// TwinCAT 3 PLC project CapSorter
// ProgramVersion: 3.1.4026.19
// libraries:
//   Tc2_Standard, * (Beckhoff Automation GmbH)
//   Tc2_System, * (Beckhoff Automation GmbH)
//   TcEventLogger, * (Beckhoff Automation Poland)
// project tree:
//   GVLs/ GVL.TcGVL, GVL_Checks.TcGVL, GVL_Communication.TcGVL, GVL_ErrorHandling.TcGVL, GVL_IO.TcGVL, GVL_Recipe.TcGVL, GVL_StandAloneUnit.TcGVL, GVL_VIS.TcGVL
//   / PlcTask.TcTTO
//   POUs/ FB_DigitalInput.TcPOU, FB_DigitalOutput.TcPOU, MAIN.TcPOU
// (motion and I/O tree: see PLC project programplc)
// real-time tasks:
//   TASK MainTask: cycle T#3ms, priority 20, ADS port 350
//   TASK SafetyTask: cycle T#10ms, priority 22, ADS port 351
//   TASK WeightTask: cycle T#2ms, priority 19, ADS port 354
//   TASK PlcTask: cycle T#10ms, priority 21, ADS port 355
//   TASK TaskToRefreshEAP: cycle T#1ms, priority 12, ADS port 301
// variable links:

CONFIGURATION CapSorter
    RESOURCE PLC ON TwinCAT3
        TASK PlcTask(INTERVAL := T#10ms, PRIORITY := 21);
        PROGRAM MAIN WITH PlcTask : MAIN;
    END_RESOURCE
END_CONFIGURATION

// ---- GVLs/GVL.TcGVL
{attribute 'qualified_only'}
VAR_GLOBAL
	iRunningMode								: INT	:= 1;					// Pozniej zastanowic sie gdzie to zostawic
END_VAR

// ---- GVLs/GVL_Checks.TcGVL
{attribute 'qualified_only'}
VAR_GLOBAL PERSISTENT
	dCheckBounds					: DINT;			// Licznik przekroczen zakresu indexow, np. tablic
	dCheckDivDInt					: DINT;			// Licznik prob dzielenia Dint przez 0
	dCheckDivLInt					: DINT; 		// Licznik prob dzielenia LInt przez 0
	dCheckDivLReal					: DINT; 		// Licznik prob dzielenia LREAL przez 0
	dCheckDivReal					: DINT; 		// Licznik prob dzielenia REAL przez 0
	dCheckRangeSigned				: DINT;			// Licznik przekroczen liczby znakowej
	dCheckRangeUnsigned				: DINT; 		// Licznik przekroczen liczby bezznakowej
END_VAR

// ---- GVLs/GVL_Communication.TcGVL
VAR_GLOBAL
//	stWrite				AT%MB0		: ST_Communication;			//Wysyłane zmienne do BottleUnboxer
//	stRead				AT%I*		: ST_Communication;			//Odczytane zmienne z BottleUnboxer

	// Sygnały pomocnicze
	bEnable									: BOOL;
	bCycleStart								: BOOL;
	bCycleStop								: BOOL;
	bCycleReset								: BOOL;
	bManualMode								: BOOL;
	bHoming									: BOOL;	
	bHomingDone								: BOOL;
	bConfectionEnding						: BOOL;	
	bHomingDialog							: BOOL;
	bHomingCanceled							: BOOL;
	bChooseRecipe							: BOOL;
	bSafetyState							: BOOL;
	bReset									: BOOL;					// reset bledow z XTS          
	bRunLock								: BOOL;					//Blokada pracy   
	bSafetyReset							: BOOL;   
	bRecipeLoading							: BOOL;					//Wystawiane jak receptura jest ładowana                                           	
	bEmptingMode							: BOOL;
	bDoorClose								: BOOL;
END_VAR

// ---- GVLs/GVL_ErrorHandling.TcGVL
{attribute 'qualified_only'}
VAR_GLOBAL
	//Zmienne obslugi bledow
	bError										: BOOL;														// Zmienna ogolna wystapienia bledu                                                                         							
	udiErrorID									: UDINT;													// Kod bledu 	
	sErrorDescription1							: STRING(200);												// Opis bledu 1
	sErrorDescription2							: STRING(200);												// Opis bledu 2
	sStationInError								: STRING(200);												// Nazwa stacji w bledzie
                                                 
                                                                        	

	tonResettingTime							: TON;														// Licznik odliczacy czas wykonywania procedury resetu
	
	iStep										: INT;														// Krok proedury czytania bledow 	

END_VAR


VAR_GLOBAL CONSTANT
	iErrorStructuresNumber						: INT					:= 9;								// Liczba strukur bledow stacji  w tym strukura bledow globalnych
END_VAR

// ---- GVLs/GVL_IO.TcGVL
VAR_GLOBAL
	
(*Wejscia DI  BC1 EK1911*)

IbPowerSupplyOK 					AT %I*		:BOOL;		//	Napięcie zasilania OK
IbDCSupply1OK 						AT %I*		:BOOL;		//	Zasilacz 10G1 OK
IbFuse10F3							AT %I*		:BOOL;		//	Blok bezpiecznikowy 10F3 OK
IbFuse10F5							AT %I*		:BOOL;		//	Blok bezpiecznikowy 10F5 OK
IbDCSupply2OK 						AT %I*		:BOOL;		//	Zasilacz 10G2 OK
ibDCSupply5VDC_OK					AT %I*		: BOOL;		// Zasilanie 5VDC OK

(* DI1 EL1008*)

IbFuseDrivesOK						AT %I*		:BOOL;		//	Zabezpieczenie Servonapędu
IbFuseTransporter					AT %I*		:BOOL;		//	Zabezpieczenie transportera modulowego
IbEmergencyStop1Active				AT %I* 		:BOOL;		//	Aktywowany przycisk zatrzymania awaryjnego Estop poniżej szafy sterowniczej
IbEmergencyStop2Active				AT %I* 		:BOOL;		//	Aktywowany przycisk zatrzymania awaryjnego Estop przy zasypie zamkniec
IbEmergencyStop3Active				AT %I* 		:BOOL;		//	Aktywowany przycisk zatrzymania awaryjnego Estop przy zasypie zamkniec	


IbSafetyDoorOpen1					AT %I*		:BOOL;		//	Otwarte drzwi 1
IbSafetyDoorOpen2					AT %I*		:BOOL;		//	Otwarte drzwi 2
QbSafetyDoorOpen					AT %Q*		:BOOL;		//	Otwarcie drzwi

(*Wyjscia DQ*)
QbResetFuse10F3						AT %Q*		:BOOL;		// Reset bloku bezpiecznikowego 10F3
QbResetFuse10F5						AT %Q*		:BOOL;		// Reset bloku bezpiecznikowego 10F5

QbBackLight							AT %Q*		:BOOL;		// Załaczenie podświetlenia koła

// Obsluga pompy prozniowej
QbVacumPumpEnable				AT %Q*		: BOOL;		// Zalaczenie pompy prozniowej
IbFuseVacumPump					AT %I*		: BOOL;		//	Zabezpieczenie pompa prozniowa	
IbVacumPumpSensor				AT %I*		: BOOL;		//Czujnik cisnienia pompa prozniowa

//Obsługa zasilania w powietrze	
IbAirSupplyOK					AT %I*		: BOOL;		// Presostat powietrza
QbAirSupply						AT %Q*		: BOOL;		// Załączanie powietrza

//Błąd działania ProfiNet
IuiProfiNetError				AT %I*		: UINT;		// Błąd komunikacji ProfiNet - 0 to OK
IuiPnIoBoxStatePickMaster		AT %I*		: UINT;		// Status komunikacji profinet
IuiPnIoBoxStateRobotABB			AT %I*		: UINT;		// Status komunikacji profinet

//Wymiana danych z robotem
QbRobotPlace1					AT %Q*		: BOOL;		// Zezwol na położenie na stlot 1 (wystawić dopiero po start w PackMlu
QbRobotPlace2					AT %Q*		: BOOL;		// Zezwol na położenie na stlot 2
QbRobotPlace3					AT %Q*		: BOOL;		// Zezwol na położenie na stlot 3
QbRobotPlace4					AT %Q*		: BOOL;		// Zezwol na położenie na stlot 4

QbRobotPlaceDoneAck1			AT %Q*		: BOOL;		// Potwierdzenie butelka odłożona 1
QbRobotPlaceDoneAck2			AT %Q*		: BOOL;		// Potwierdzenie butelka odłożona 2
QbRobotPlaceDoneAck3			AT %Q*		: BOOL;		// Potwierdzenie butelka odłożona 3
QbRobotPlaceDoneAck4			AT %Q*		: BOOL;		// Potwierdzenie butelka odłożona 4

QbRobotStepMode					AT %Q*		: BOOL;		// Praca krokowa

QbRobotService					AT %Q*		: BOOL;		// Przejście robota w tryb serwisowy - potrzebne do ManualMovements
{warnin: DO usuniecia}
QbRobotServicePlace1			AT %Q*		: BOOL;		// Ruch robota do stlot 1 
QbRobotServicePlace2			AT %Q*		: BOOL;		// Ruch robota do stlot 2
QbRobotServicePlace3			AT %Q*		: BOOL;		// Ruch robota do stlot 3
QbRobotServicePlace4			AT %Q*		: BOOL;		// Ruch robota do stlot 4

QbRobotServiceVacumOn			AT %Q*		: BOOL;		// Załącz vacum
QbRobotServiceRejectOn			AT %Q*		: BOOL;		// Załącz odrzut
{warnin: DO usuniecia}
QbRobotServiceGripper			AT %Q*		: BOOL;		// Pozycja ramienia
{warnin: DO usuniecia}
IbRobotQueueFull1				AT %I*		: BOOL;		// Butelka wyjęta z kolejki wykrytych (nie wiem po co to nam)
IbRobotQueueFull2				AT %I*		: BOOL;		// Butelka wyjęta z kolejki wykrytych (nie wiem po co to nam)
IbRobotQueueFull3				AT %I*		: BOOL;		// Butelka wyjęta z kolejki wykrytych (nie wiem po co to nam)

IbRobotPlaceDone1				AT %I*		: BOOL;		// Butelka odłożona 1
IbRobotPlaceDone2				AT %I*		: BOOL;		// Butelka odłożona 2
IbRobotPlaceDone3				AT %I*		: BOOL;		// Butelka odłożona 3
IbRobotPlaceDone4				AT %I*		: BOOL;		// Butelka odłożona 4
{warnin: DO usuniecia}
IbRobotPosAvailable1			AT %I*		: BOOL;		// Potwierdzenie przyjęcia pozycji Place1
IbRobotPosAvailable2			AT %I*		: BOOL;		// Potwierdzenie przyjęcia pozycji Place2
IbRobotPosAvailable3			AT %I*		: BOOL;		// Potwierdzenie przyjęcia pozycji Place3

IbRobotVacumOn					AT %I*		: BOOL;		//Sygnał załaczenia Vacum
IbRobotVacumLevelOk				AT %I*		: BOOL;		//Sygnał z czujnika Vacum

IbRobotAutoOn					AT %I*		: BOOL;
IbRobotEmmergencyStop			AT %I*		: BOOL;
IbRobotExecutionError			AT %I*		: BOOL;
IbRobotMotionSupTrig			AT %I*		: BOOL;		// Kolizja
IbRobotMotorsOnState			AT %I*		: BOOL;
IbRobotRevCounterLost			AT %I*		: BOOL;		//Brak kalibracji
IbRobotTaskExecuting			AT %I*		: BOOL;		//Program się wykonuje
IbRobotWriteAcces				AT %I*		: BOOL;		//Załaczony dostęp zdalny
IbRobotSMBBatteryChargeLow		AT %I*		: BOOL;		//Alarm baterii


IdiRobotUnitModeCurrent			AT %I*		: DINT;	
IdiRobotStateCurrent			AT %I*		: DINT;	
IdiRobotRobotStatus0			AT %I*		: INT;
IdiRobotRobotStatus1			AT %I*		: INT;
IbRobotRobotIdle				AT %I*		: BOOL;
IbRobotRobotError				AT %I*		: BOOL;
IbRobotRobotPMRTConnected		AT %I*		: BOOL;
IbRobotRobotHeartBeat			AT %I*		: BOOL;
IudiRobotActiveOrder			AT %I*		: UDINT;	
IudiRobotErrorCode				AT %I*		: UDINT;	
IudiRobotCurrentRecipeID		AT %I*		: UDINT;	
IdiRobotBottelsCount			AT %I*		: DINT;
IuiRobotFieldbusType			AT %I*		: UINT := 2;

QdiRobotUnitMode				AT %Q*		: DINT;	
QdiRobotCntrlCmd				AT %Q*		: DINT;	
QdiRobotRobotCmd0				AT %Q*		: INT;
QdiRobotRobotCmd1				AT %Q*		: INT;
QbRobotUnitModeChangeRequest	AT %Q*		: BOOL;	
QbRobotCmdChangeRequest			AT %Q*		: BOOL;	
QbRobotRequest					AT %Q*		: BOOL;	
QbRobotResetError				AT %Q*		: BOOL;	
QudiRobotRequestOrder			AT %Q*		: UDINT;	
QudiRobotRequestRecipeID		AT %Q*		: UDINT;	

QbRobotGetFlowCount				AT %Q*		: BOOL;

QbEmptingDoorSolenoid			AT %Q*		: BOOL;

END_VAR

// ---- GVLs/GVL_Recipe.TcGVL
(*
Nazwa:			GVL_Recipe
Opis:			Zmienne recepturowe tylko do wizualizacji
Wersja:			v0.2
Data:			2024-02-20
Autor:			MK
Urzadzenia:		
Konfiguracja:	
Info:
Zmiany:
- 20240220 [DP] Poprawki przed nowa wizką
*)
VAR_GLOBAL
	(*Legenda dla wizki :
		[H] - Hidden, prawdopodobnie nie potrzebne
		[I] - Info, informacja,
		[L] - Later, do zrobienia później, być może do przerobienia
		Uprawienia:
		brak opisu - operator
		[m] - Meechanik i powyżej
		[t] - Technolog i powyżej
		[s] - Serwis i powyżek
		[a] - Admin			
	*)	
	
	//Sorter nasadek, typ produktu	
	iCapSorterProductType										: INT		:= 2; 		//		Typ produktu: 0- kule/fliptopy, 1- pompki, 2- disctop, 3-airless, 4-decoration cap (wyłączone podcisnienie na załapywarce), 5- decoration cap with new gripper (wyłączone podcisnienie + nowy program do robota)
	uiCapSorterIndexShow										: UDINT		:= 5;		//		Index produktu	
	bPresenceBottleEnableShow									: BOOL;					//		Sprawdzanie butelki w formatce

//--------------------------------------CapSorterTransporter-----------------------------------------------------------------------------------------------------------------------------	
	// Sorter nasadek, transporter zasobnika
	bCapSorterTransporterEnableShow								: BOOL;					//		Aktywacja
	iCapSorterTransporterTankConveyorVelocityShow				: INT		:= 1200;	//		Prędkość 							| [%] (1.0-100.0)
	iCapSorterTransporterStartDelayTimeShow						: INT		:= 100;		//		Timer do załączania 				| [ms] (0.0-10_000.0)
	udiCapSorterTransporterTimeProductOnSensorBeforeBrushShow	: UDINT		:= 150;		//		Timer pracy							| [ms] (0.0-10_000.0)
	iCapSorterTransporterEmptyingConveyorSpeedShow				: INT		:= 25;		// 		Prędkość, opróżnianie 				| [%] (1.0-100.0)
	iCapSorterTransporterVolumeOfCapsShow						: INT		:= 330;		//		Odłegłość do zamknięć, ostrzeżenie 	| [mm] (0.0-10_000.0)

//---------------------------------------CapSorterWheel----------------------------------------------------------------------------------------------------------------------------	
	// Sorter nasadek, stól
	bCapSorterWheelEnableShow									: BOOL;					//		Aktywacja
	lrCapSorterWheelMoveAccelerationEmptyTableShow				: LREAL		:= 5000;	//		Dynamika rozpędzania - pusty 		| [obr/min²], (1.0-100_000.0) 
	lrCapSorterWheelMoveDecelerationEmptyTableShow				: LREAL		:= 5000;    //		Dynamika spowalniania - pusty 		| [obr/min²] (1.0-100_000.0) 
	lrCapSorterWheelMoveSpeedEmptyTableShow						: LREAL		:= 334;     //		Prędkość - pusty 					| [obr/min] (1.0-10_000.0)                
	lrCapSorterWheelMoveAngleEmptyTableShow						: LREAL		:= 20;      //		Kąt - pusty 						| [obr/min] (0.0-360.0)                        
	lrCapSorterWheelJerkAngleEmptyTableShow						: LREAL		:= 15000;   //		Zryw - pusty 						| [obr/min³] (1.0-1_000_000)                  
	iCapSorterWheelWaitingAfterRotationEmptyTableShow			: INT		:= 100;     //		Czas stabilizacji - pusty 			| [ms] (0.0-1_000)                 
	
	lrCapSorterWheelMoveAccelerationFullTableShow				: LREAL		:= 5000;	//		Dynamika rozpędzania - pełny 		| [obr/min²], (1.0-100_000.0) 
	lrCapSorterWheelMoveDecelerationFullTableShow				: LREAL		:= 5000;    //		Dynamika spowalniania - pełny 		| [obr/min²] (1.0-100_000.0) 
	lrCapSorterWheelMoveSpeedFullTableShow						: LREAL		:= 334;     //		Prędkość - pełny 					| [obr/min] (1.0-10_000.0)                
	lrCapSorterWheelMoveAngleFullyTableShow						: LREAL		:= 6;       //		Kąt - pełny 						| [obr/min] (0.0-360.0)                        
	lrCapSorterWheelJerkAngleFullTableShow						: LREAL		:= 15000;   //		Zryw - pełny 						| [obr/min³] (1.0-1_000_000)                  
	iCapSorterWheelWaitingAfterRotationFullTableShow			: INT		:= 30;      //		Czas stabilizacji - pełny 			| [ms] (0.0-1_000)                 
	
	lrCapSorterWheelMoveAccelerationHalfFullTableShow			: LREAL		:= 5000;	//		Dynamika rozpędzania - półpełny 	| [obr/min²], (1.0-100_000.0) 
	lrCapSorterWheelMoveDecelerationHalfFullTableShow			: LREAL		:= 5000;    //		Dynamika spowalniania - półpełny 	| [obr/min²] (1.0-100_000.0) 
	lrCapSorterWheelMoveSpeedHalfFullTableShow					: LREAL		:= 334;     //		Prędkość - półpełny 				| [obr/min] (1.0-10_000.0)                
	lrCapSorterWheelMoveAngleHalfFullyTableShow					: LREAL		:= 12;      //		Kąt - półpełny						| [obr/min] (0.0-360.0)                        
	lrCapSorterWheelJerkAngleHalfFullTableShow					: LREAL		:= 15000;   //		Zryw - półpełny 					| [obr/min³] (1.0-1_000_000)                  
	iCapSorterWheelWaitingAfterRotationHalfFullTableShow		: INT		:= 50;      //		Czas stabilizacji - półpełny 		| [ms] (0.0-1_000)               
	
//-------------------------------------CapSorterCamera------------------------------------------------------------------------------------------------------------------------------	                                                    	
	// Sorter nasadek, system wizyjny
	
    bCapSorterCameraEnableShow									: BOOL; 				//	[H]	Aktywacja                            	
	
//-----------------------------------------CapSorterRobot--------------------------------------------------------------------------------------------------------------------------	
	// Sorter nasadek, robot
	bCapSorterRobotEnableShow									: BOOL;					//		Aktywacja
                                                                                                                           	
	lrCapSorterRobotPlace1PositionXShow							: LREAL;				//		Offset odkładania 1, X 			| [mm]	((-100.0)-100.0)       
	lrCapSorterRobotPlace1PositionYShow							: lreal;    			//		Offset odkładania 1, Y 			| [mm]	((-100.0)-100.0)       
	lrCapSorterRobotPlace1PositionZShow							: lreal;    			//		Offset odkładania 1, Z 			| [mm]	((-100.0)-100.0)       
	lrCapSorterRobotPlace1PositionCShow							: lreal;    			//		Offset odkładania 1, C 			| [° ]	((-360.0)-360.0)                 
	iCapSorterRobotPickElevationShow							: INT;					//		Punkt nad poz. Pick				| [mm]	(30-1000)
	iCapSorterRobotPickTimeShow									: INT;					//		Czas przyssania					| [ms]	(0-10_000)
	iCapSorterRobotVacuumActivationShow							: INT;					//		Czas przed przyssaniem			| [ms]	(0-1000)
	iCapSorterRobotVacuumOffShow								: INT;					//		Czas przed oddmuchem			| [ms]	(0-1000)
	iCapSorterRobotPlaceTimeShow								: INT;					//		Czas oddmuchu					| [ms]	(0-1000)
	iCapSorterRobotTCP_PlaceOffsetShow							: INT;					//		Wysokość od TCP do p. odłożenia	| [mm]	(0-1000)									
	iCapSorterRobotAccelerationDecelerationShow					: INT;					//		Dynamika rozpędzania/hamowania	| [%]	(20-100)
	iCapSorterRobotGripperWatchdogShow							: INT;					//		Czas sprawdzania silownika		| [ms]	(0-1000)
	iCapSorterRobotParalaxCorrectionShow						: INT;					//		Korekta paralaxy				| [mm]	(0-100)
	
	iCapSorterRobotNumberToolShow								: INT;					//		Numer narzędzia					| 		(0-10)
	iCapSorterRobotPickPositionZShow							: INT;					//		Wysokość pobierania 			| [mm]	(0-200)
	iCapSorterRobotTCP_Lenght									: INT;					//		Długość chwytaka				| [mm]	(10-100)
	iCapSorterRobotProductDiametr								: INT;					//		Średnica nasadki				| [mm] 	(10-100)
	
//----------------------------------------CapSorterIntermediateTransporter---------------------------------------------------------------------------------------------------------------------------
	// Sorter nasadek, transporter zasypowy
	bCapSorterIntermediateTransporterEnableShow					: BOOL;					//		Aktywacja
	iCapSorterIntermediateTransporterAutoSpeedShow				: INT		:= 20;		//		Prędkość 					| [%] (1.0-100.0)
	iCapSorterIntermediateTransporterManualSpeedShow			: INT		:= 30;		//		Prędkość, manual 			| [%] (1.0-100.0)
	iCapSorterIntermediateTransporterEmptyingSpeedShow			: INT		:= 50;		//		Prędkość, opróżnianie 		| [%] (1.0-100.0)
	iCapSorterIntermediateTransporterDelayCountTimeShow			: INT		:= 100;		//		Timer pracy					| [ms]	(0.0-100_000.0)
	iCapSorterIntermediateTransporterReverseTimeShow			: INT		:= 4000;	//		Timer odwróconej pracy 		| [ms] (0.0-10_000.0)
	udiCapSorterIntermediateTransporterTimeProductOnSensorShow	: UDINT		:= 1800;	//		Czas produktu na czujniku 	| [ms] (0.0-10_000.0)	
	lrCapSorterIntermediateTransporterWheelAngleShow			: LREAL		:= 6;		//		Kąt zasypu 					| [°] (1.0-360.0)
	lrCapSorterIntermediateTransporterItemsSetValueShow			: LREAL	;				// 		Ilość detali na kołe		| []
	
//----------------------------------------CapSorterIntermediateBrush---------------------------------------------------------------------------------------------------------------------------
	//Sorter nasadek, szczotka transportera
	bCapSorterIntermediateBrushEnableShow						: BOOL;					//		Aktywacja
	iCapSorterIntermediateBrushAutoSpeedShow					: INT		:= 30;		//		Prędkość  					| [%] (0.0-100.0)
	iCapSorterIntermediateBrushManualSpeedShow					: INT		:= 30;		//		Prędkość, manual 			| [%] (0.0-100.0)
	iCapSorterIntermediateBrushEmptyingSpeedShow				: INT		:= 30;		//		Prędkość, opróżnianie 		| [%] (0.0-100.0)
	lrCapSorterIntermediateBrushPositionHeightSVShow			: LREAL		:= 45;		//		Wysokość 					| [mm] (0.0-10_000.0)

//----------------------------------------CapSorterBrush1OnWheel---------------------------------------------------------------------------------------------------------------------------
	// Sorter nasadek, szczotka stolu 1
	bCapSorterBrush1OnWheelEnableShow							: BOOL;					//		Aktywacja
	iCapSorterBrush1OnWheelAutoSpeedShow						: INT		:= 30;		//		Prędkość 					| [%] (0.0-100.0)
	iCapSorterBrush1OnWheelManualSpeedShow						: INT		:= 30;		//		Prędkość, manual 			| [%] (0.0-100.0)
	iCapSorterBrush1OnWheelEmptyingSpeedShow					: INT		:= 30;		//		Prędkość, opróżnianie 		| [%] (0.0-100.0)
	lrCapSorterBrush1OnWheelPositionHeightSVShow				: LREAL		:= 45;		//		Wysokość 					| [mm] (0.0-10_000.0)
	
//----------------------------------------CapSorterBrush2OnWheel----------------------------------------------------------------------------------
	// Sorter nasadek, szczotka stolu 2
	bCapSorterBrush2OnWheelEnableShow							: BOOL;					//		Aktywacja
	iCapSorterBrush2OnWheelAutoSpeedShow						: INT		:= 30;		//		Prędkość 					| [%] (0.0-100.0)
	iCapSorterBrush2OnWheelManualSpeedShow						: INT		:= 30;		//		Prędkość, manual 			| [%] (0.0-100.0)
	iCapSorterBrush2OnWheelEmptyingSpeedShow					: INT		:= 30;		//		Prędkość, opróżnianie 		| [%] (0.0-100.0)
	lrCapSorterBrush2OnWheelPositionHeightSVShow				: LREAL		:= 45;		//		Wysokość 					| [mm] (0.0-10_000.0)

//------------------------------------------CapFeeder-------------------------------------------------------------------------------------------------------------------------	
	// Sorter nasadek, 
	bCapSorterFeederEnableShow									: BOOL;					//		Aktywacjaa
	bCapSorterFeederEnableTubeError								: BOOL;					// 		Aktywacja błedu słomki
	lrCapSorterFeederMover1InputPositionShow					: LREAL;				//		Pozycja wkładania, wózek 1 	| [mm] (?-?)
	lrCapSorterFeederMover2InputPositionShow					: LREAL;				//		Pozycja wkładania, wózek 2 	| [mm] (?-?)
	lrCapSorterFeederMover1OutputPositionShow					: LREAL;				//		Pozycja wyjmowania, wózek 1 | [mm] (?-?)
	lrCapSorterFeederMover2OutputPositionShow					: LREAL;				//		Pozycja wyjmowania, wózek 2 | [mm] (?-?)
	lrCapSorterFeederSlotDistanceShow							: LREAL;				//		Offset wkładania			| [mm] (?-?)			Old-(Odstęp między pozycjami kładzenia)
	lrCapSorterFeederMoverSpeedShow								: LREAL;				//		Prędkość				 	| [%] (0.0-100.0)
	lrCapSorterFeederMoverAccelerationShow						: LREAL;				//		Przyspieszenie 				| [mm/s²] 
	lrCapSorterFeederMoveJerkShow								: LREAL;				//		Zryw						| [mm/s³]

//-------------------------------------------------------------------------------------------------------------------------------------------------------------------	
	//CapPreScrewer		
	bCapSorterPreScrewerEnableShow								: BOOL;					// 		Aktywacja
	bCapSorterPreScrewerPicker1EnableShow						: BOOL;					// 		Aktywacja	
	bCapSorterPreScrewerPicker2EnableShow						: BOOL;					// 		Aktywacja
	bCapSorterPreScrewerPicker3EnableShow						: BOOL;					// 		Aktywacja	
	bCapSorterPreScrewerPicker4EnableShow						: BOOL;					// 		Aktywacja
	//Oś Z
	lrCapSorterPreScrewerPickZPositionShow						: LREAL;				//		Wysokość pobierania						| [mm]	
	lrCapSorterPreScrewerCatcherReleseShow						: LREAL;				//		nie używamy Wysokość otwierania chwytaka nakrętek	| [mm]		
	lrCapSorterPreScrewerCapCatcherZPositionShow				: LREAL;				//		Wysokość zamykania nakrętkek			| [mm]
	lrCapSorterPreScrewerTopZPositionShow						: LREAL;				//		Pozycja górna ośi Z						| [mm] 	
	lrCapSorterPreScrewerCartesianCatchZPositionShow			: LREAL; 				//      Wait Position
	lrCapSorterPreScrewerStrawCatcherZPositionShow				: LREAL;				//		Wysokość otwierania łapaczy słomek		| [mm]	
	LrCapSorterPreScrewerCheckStrawCatcherActuatorZPosition		: LREAL;				//		Wysokość sparawdzania cofania łapaczy słomek	| [mm]	
	lrCapSorterPreScrewerScrewerStartZPositionShow				: LREAL;				//		Wysokość początku zakręcania			| [mm]	
	lrCapSorterPreScrewerGripperOpenPositionShow				: LREAL;				//		Pozycja otwierania chwytaka butelek 	| [mm]
	lrCapSorterPreScrewerPlaceZPositionShow						: LREAL;				//		Wysokość odkładania - koniec załapywania gwintu	| [mm] 

	lrCapSorterPreScrewerThreadPitchShow						: LREAL;				//		Skok gwintu 		| [mm]	
	lrCapSorterPreScrewerMultipleStartThreadShow				: LREAL;				//		Krotność gwintu
	lrCapSorterPreScrewerNumberOfThreadTurnsShow				: LREAL;				//		Ilość obrotów
  	
	//Wspólne ruchi	
	lrCapSorterPreScrewerBendingDistanceShow					: LREAL;				//		Odległość zaokrąglania ruchów 			| [mm]		
	lrCapSorterPreScrewerStrawInsertDistance					: LREAL;				//		Odległość wspólnego ruchu, prowadzenie słomki	| [mm]		
	//Oś x
	lrCapSorterPreScrewerPickXMover1PositionShow				: LREAL;				//		Pozycja osi poziomej do pobierania, wozek 1	| [mm]
	lrCapSorterPreScrewerPickXMover2PositionShow				: LREAL;				//		Pozycja osi poziomej do pobierania, wozek 2	| [mm]
	lrCapSorterPreScrewerPlaceXPositionShow						: LREAL;				//		Pozycja osi poziomej do odkładania			| [mm]
	//Oś zakręcania
	lrCapSorterPreScrewerScrewFindingShow						: LREAL;				//		Kąt szukania gwintu							| [°]
	lrCapSorterPreScrewerScrewDistanceShow						: LREAL;				//		Kąt zakręcania								| [°]
	//Prédkośći                                                                                                                         	
	lrCapSorterPreScrewerPickerSpeedShow						: LREAL;				//		Prędkość									| [%]   
	lrCapSorterPreScrewerPickerSpeedWhenScrewerShow				: LREAL;				//		Prędkość osi Z przy zakręcaniu				| [%]   
	lrCapSorterPreScrewerPickerAccelerationShow					: LREAL;				//		Przyspieszenie								| [mm/s²] 		
	lrCapSorterPreScrewerPickerJerkShow							: LREAL;				//		Zryw										| [mm/s³]
                                                                                                                                        	
	lrCapSorterPreScrewerCatcherSpeedShow						: LREAL;				//		Prędkość									| [mm/s] 
	lrCapSorterPreScrewerCatcherAccelerationShow				: LREAL;				//		Przyspieszenie								| [mm/s²] 	
	lrCapSorterPreScrewerCatcherJerkShow						: LREAL;				//		Zryw										| [mm/s³]	                                                                                                                                 	
	lrCapSorterPreScrewerScrewSpeedShow							: LREAL;				//		Prędkość zakręcania							| [mm/s]
	lrCapSorterPreScrewerScrewAccelerationShow					: LREAL;				//		Przyspieszenie zakręcania				| [mm/s²]
	lrCapSorterPreScrewerScrewJerkShow							: LREAL;				//		Zryw zakręcania							| [mm/s³]

	//Oś łapacza słomki	
	lrCapSorterPreScrewerCatcherCatchingPositionShow			: LREAL;				//		Pozycja łapania słomki					| [mm]
	lrCapSorterPreScrewerCatcherPlacePositionShow				: LREAL;				//		Pozycja dolna łapacza słomki			| [mm]
	lrCapSorterPreScrewerCatcherHightSVShow						: LREAL;				//		Nastawa wysokości stacji łapacza słomek		| [mm]
	//Kalibracja chwytaków butelki
	bCapSorterPreScrewerBottleCatcherEnableShow					: BOOL;					//		Actywacja chwytaków butelki
	lrCapSorterPreScrewerBottleCatch1OpenValueShow				: LREAL;				//		Chwytak 1 | wartość kalibracji otwartego chwytaka
	lrCapSorterPreScrewerBottleCatch1CloseValueShow				: LREAL;				//		Chwytak 1 | wartośc kalibracji zamkniętego chwytaka
	lrCapSorterPreScrewerBottleCatch2OpenValueShow				: LREAL;				//		Chwytak 2 | wartość kalibracji otwartego chwytaka
	lrCapSorterPreScrewerBottleCatch2CloseValueShow				: LREAL;				//		Chwytak 2 | wartość kalibracji zamkniętego chwytaka
	lrCapSorterPreScrewerBottleCatch3OpenValueShow				: LREAL;                //		Chwytak 3 | wartość kalibracji otwartego chwytaka
	lrCapSorterPreScrewerBottleCatch3CloseValueShow				: LREAL;				//		Chwytak 3 | wartość kalibracji zamkniętego chwytaka	
	lrCapSorterPreScrewerBottleCatch4OpenValueShow				: LREAL;                //		Chwytak 4 | wartość kalibracji otwartego chwytaka
	lrCapSorterPreScrewerBottleCatch4CloseValueShow				: LREAL;				//		Chwytak 4 | wartość kalibracji zamkniętego chwytaka
	                                                        	
	lrCapSorterPreScrewerBottleCatchToleranceValueShow			: LREAL;				//		Tolerancja chwytaków
	lrCapSorterPreScrewerCatchAngleOpenSV						: LREAL := 180.0;		//		[] Kąt puszczania centrowników
	
	lrCapSorterPreScrewerWaitInPlaceTimeShow					: LREAL	:= 50;			//		Czas zatrzymania w miejscu odłożenia 	| [ms]
	
	bCapSorterPreScrewerCatchAngleOpenEnaShow					: BOOL;					// 		Aktywacja puszczania centrowników po osiągnięciu zadanego kątu
	bCapSorterPreScrewerPoundedInCap							: BOOL;					// 		Wbijana nasadka
	
//Parametry do obliczeń 
	lrCapSorterBottleHightShow									: LREAL;				//		Wysokość butelki
	lrCapSorterBottleNeckHightShow								: LREAL;				// 		Wysokość szyjki butelki
	lrCapSorterCapHightShow										: LREAL;				// 		Wysokość zamknięcia
	lrCapSorterCapNeckHightShow									: LREAL;				//		Wysokość szyjki zamknięcia
	lrCapSorterPreScrewerCheckValveShow							: LREAL;				//		Długość zaworu zwrotnego				| [mm]
	
	lrCapSorterMoverHightShow									: LREAL := 226.0;		//		Wysokość wózków (Kartezjanem dotknąć ssawkami gniazdo do wkładania zamknięć)
	
//Rezerwa	
	lrCapSorterSpare1											: LREAL;				//Rezerwa 1
	lrCapSorterSpare2											: LREAL;				//Rezerwa 2
	lrCapSorterSpare3											: LREAL;				//Rezerwa 3
	lrCapSorterSpare4											: LREAL;				//Rezerwa 4
	lrCapSorterSpare5											: LREAL;				//Rezerwa 5
	lrCapSorterSpare6											: LREAL;				//Rezerwa 6
	lrCapSorterSpare7											: LREAL;				//Rezerwa 7	
	
	
	
END_VAR

// ---- GVLs/GVL_StandAloneUnit.TcGVL
{attribute 'qualified_only'}
VAR_GLOBAL
	bStandAlone									: BOOL;		// Without superior system
	bNoPackML									: BOOL;		// Without PackML
	bGhostMode									: BOOL; 	// Without product, demo mode
	bStartCycle									: BOOL;
	bStopCycle									: BOOL;
	bServiceMode								: BOOL;
	bHoming										: BOOL;
	bReset										: BOOL;
	bChooseRecipe								: BOOL;
	bProductionEnding							: BOOL;
	bDoorOpen									: BOOL;
	
END_VAR

// ---- GVLs/GVL_VIS.TcGVL
(*
Nazwa:			GVL_VIS
Opis:			Zmienne dla wizualizacji
Wersja:			v0.2
Data:			2024-02-20
Autor:			AS
Urzadzenia:		
Konfiguracja:	
Info:
Zmiany:
- 20240220 [DP] Poprawki przed nowa wizką
*)

{attribute 'qualified_only'}
VAR_GLOBAL	
(*
Nazwa:			GVL_VIS
Opis:			Zmienne dla wizualizacji
Wersja:			v0.2
Data:			2024-02-20
Autor:			MK
Urzadzenia:		
Konfiguracja:	
Info:
Zmiany:
- 20240220 [DP] Poprawki przed nowa wizką
*)

//-----------------------------------------CapSorterWheel--------------------------------------------------------------------------------------------------------------------------	
	//Sorter nasadek, koło
	iCapSorterWheelState							: INT;				// Stan
	sCapSorterWheelState							: STRING;   		// Stan
	bCapSorterWheelHoming							: BOOL;             // Bazowanie					// Przycisk bistabilny                     Bazowanie                                       									
	bCapSorterWheelManualWheelRight    				: BOOL;   			// Do przodu					// Przycisk monostabilny                     						
	bCapSorterWheelManualWheelLeft     				: BOOL;  			// Do tyłu						// Przycisk monostabilny  						
	bCapSorterWheelManualContinuousMovement			: BOOL;				// obrót o zadany kąt			// Przycisk bistabilny					
                                                                                               
//-----------------------------------------CapSorterCamera--------------------------------------------------------------------------------------------------------------------------	
	//Sorter nasadek, system wizyjny
	iCapSorterCameraState							: INT;				// Stan
	sCapSorterCameraState							: STRING;			// Stan
	bCapSorterCameraHoming							: BOOL;				// Bazowanie					// Przycisk bistabilny    	                                                	
	bCapSorterCameraManualRun						: BOOL;				// Zrób zdięcie					// Przycisk monostabilny
	bCapSorterBacklightManualStart					: BOOL;				// Podświetlenie stolu			// Przycisk bistabilny  
	uiCapSorterCameraActualJobIDLoaded				: UDINT;   	        // Program załadowany			// Pole do wyświetlania wartości                                   
	lrCapSorterCameraPickPointXVisu					: LREAL;			// Współrzędne produktu, X		// Pole do wyświetlania wartości
	lrCapSorterCameraPickPointYVisu					: LREAL;			// Współrzędne produktu, Y		// Pole do wyświetlania wartości
	lrCapSorterCameraPickPointAngleVisu				: LREAL;			// Kąt produktu					// Pole do wyświetlania wartości
                                                 	
//------------------------------------------ CapSorterRobot-------------------------------------------------------------------------------------------------------------------------	
	//Sorter nasadek, robot
	iCapSorterRobotState							: INT;				// Stan
	sCapSorterRobotState							: STRING;           // Stan
	bCapSorterRobotHoming							: BOOL;             // Bazowanie					// Przycisk bistabilny                                	
	
	bCapSorterRobotManualSuction					: BOOL; 			// Ssawka						// Przycisk bistabilny
	bCapSorterRobotManualGripperArmPosition1		: BOOL;  			// Ramię robota					// Przycisk bistabilny	
	bCapSorterRobotReadyPosition 					: BOOL;     		// Gotowość                                                                  	
	bCapSorterRobotPreparePick 						: BOOL;     		// Przygotuj do pobrania	
	bCapSorterRobotPick 							: BOOL;     		// Pobierz						// Przycisk bistabilny
	bCapSorterRobotPreparePlace						: BOOL;     		// Przygotuj do odłożenia
	bCapSorterRobotPlace							: BOOL;     		// Odłóż						// Przycisk bistabilny
	diCapSorterRobotPlaceId							: DINT; 			// Slot odłożenia | (1-4) 		// Pole do wpisywania wartosci
	diCapSorterRobotSpeed							: DINT; 			// Prędkość | [%] (1-100)		// Pole do wpisywania wartosci

		
//----------------------------------CapSorterTransporter---------------------------------------------------------------------------------------------------------------------------------
	//Sorter nasadek, transporter zasobnika
	iCapSorterTransporterState						: INT;				// Stan
	sCapSorterTransporterState						: STRING;           // Stan
	bCapSorterTransporterHoming						: BOOL;		        // Bazowanie					// Przycisk bistabilny                                          	
	bCapSorterTransporterManualTankConveyor			: BOOL;       		// Do przodu					// Przycisk bistabilny
	bCapSorterTransporterManualTankConveyorRevers	: BOOL;             // Do tyłu						// Przycisk bistabilny                                   	                                           	
		
	
	
//----------------------------------------CapSorterIntermediateTransporter---------------------------------------------------------------------------------------------------------------------------	
	// Sorter nasadek, transporter zasypowy
	iCapSorterIntermediateTransporterState			: INT;				// Stan
	sCapSorterIntermediateTransporterState			: STRING;	        // Stan                                      
	bCapSorterIntermediateTransporterHoming			: BOOL;             // Bazowanie					// Przycisk bistabilny   
	bCapSorterIntermediateTransporterManualForward	: BOOL;             // Do przodu					// Przycisk bistabilny
	bCapSorterIntermediateTransporterManualBackward	: BOOL;				// Do tyłu						// Przycisk bistabilny   
	
//----------------------------------------CapSorterIntermediateBrush---------------------------------------------------------------------------------------------------------------------------	
	//Sorter nasadek, szczotka transportera
	iCapSorterIntermediateBrushState				: INT;	  			// Stan
	sCapSorterIntermediateBrushState				: STRING;           // Stan
	bCapSorterIntermediateBrushHoming				: BOOL;             // Bazowanie					// Przycisk bistabilny                                      
	bCapSorterIntermediateBrushWeightSet			: BOOL;				// Ustaw pozycje				// Przycisk bistabilny
	bCapSorterIntermediateBrushManualForward		: BOOL;             // Do przodu					// Przycisk bistabilny
	bCapSorterIntermediateBrushManualBackward		: BOOL;		        // Do tyłu						// Przycisk bistabilny                                           
	bCapSorterIntermediateBrushManualLiftUp			: BOOL;				// Do góry						// Przycisk monostabilny
	bCapSorterIntermediateBrushManualLiftDown		: BOOL;             // Do dołu						// Przycisk monostabilny
	lrCapSorterIntermediateBrushActualHeight		: LREAL;			//Aktualna wysokosc | [mm]				// Pole do wyświetlania wartości
		
//-------------------------------------------CapSorterBrush1------------------------------------------------------------------------------------------------------------------------
	// Sorter nasadek, szczotka stolu 1
	iCapSorterBrush1OnWheelState					: INT;				// Stan
	sCapSorterBrush1OnWheelState					: STRING;           // Stan
	bCapSorterBrush1OnWheelHoming					: BOOL;	            // Bazowanie					// Przycisk bistabilny                                                       
	bCapSorterBrush1WeightSet						: BOOL;				// Ustaw pozycje				// Przycisk bistabilny
	bCapSorterBrush1OnWheelManualLiftUp				: BOOL;             // Do przodu					// Przycisk bistabilny
	bCapSorterBrush1OnWheelManualLiftDown			: BOOL;	            // Do tyłu						// Przycisk bistabilny                                                       
	bCapSorterBrush1OnWheelManualDriveForward		: BOOL;             // Do góry						// Przycisk monostabilny
	bCapSorterBrush1OnWheelManualDriveBackward		: BOOL;             // Do dołu						// Przycisk monostabilny
	lrCapSorterBrush1OnWheelActualHeight			: LREAL;	        //Aktualna wysokosc | [mm]				// Pole do wyświetlania wartości
	
//----------------------------------------CapSorterBrush2---------------------------------------------------------------------------------------------------------------------------	
	// Sorter nasadek, szczotka stolu 2
	iCapSorterBrush2State							: INT;				// Stan
	sCapSorterBrush2State							: STRING;           // Stan
	bCapSorterBrush2Homing							: BOOL;	            // Bazowanie					// Przycisk bistabilny                   
	bCapSorterBrush2WeightSet						: BOOL;				// Ustaw pozycje				// Przycisk bistabilny	
	bCapSorterBrushManualBrush2OnWheelLiftUp		: BOOL;             // Do przodu					// Przycisk bistabilny
	bCapSorterBrushManualBrush2OnWheelLiftDown		: BOOL;             // Do tyłu						// Przycisk bistabilny                   
	bCapSorterBrushManualBrush2OnWheelDriveForward	: BOOL;             // Do góry						// Przycisk monostabilny
	bCapSorterBrushManualBrush2OnWheelDriveBackward	: BOOL;             // Do dołu						// Przycisk monostabilny
	lrCapSorterBrush2OnWheelActualHeight			: LREAL;            //Aktualna wysokosc | [mm]				// Pole do wyświetlania wartości		

//-------------------------------------------------------------------------------------------------------------------------------------------------------------------	
	//Sorter nasadek, CapFeeder
	iCapSorterFeederState							: INT;			// Stan
	lrCapSorterFeederMover1CVShow					: LREAL;		// Pozycja mówera 1
	lrCapSorterFeederMover2CVShow					: LREAL;		// Pozycja mówera 2  
	sCapSorterFeederState							: STRING;       // Stan
	bCapSorterFeederHoming							: BOOL;			// Bazowanie						// Przycisk bistabilny 
	bCapSorterFeederMover1Forvard 					: BOOL;			// Mover 1 +						// Przycisk monostabilny
	bCapSorterFeederMover1Backward					: BOOL;			// Mover 1 -						// Przycisk monostabilny
	bCapSorterFeederMover2Forvard 					: BOOL;			// Mover 2 +						// Przycisk monostabilny
	bCapSorterFeederMover2Backward					: BOOL;			// Mover 2 -						// Przycisk monostabilny
	bCapSorterFeederMover1ActuatorIn				: BOOL;			// Mover 1 Do przodu				// Przycisk bistabilny
	bCapSorterFeederMover1ActuatorOut				: BOOL;			// Mover 1 Do tyłu					// Przycisk bistabilny
	bCapSorterFeederMover1PickPos					: BOOL;			// Mover 1, pozycja pobrania		// przycisk monostabilny
	bCapSorterFeederMover1PlacePos					: BOOL;			// Mover 1, pozycja odkładania		// przycisk monostabilny
	bCapSorterFeederMover2PickPos					: BOOL;			// Mover 2, pozycja pobrania		// przycisk monostabilny
	bCapSorterFeederMover2PlacePos					: BOOL;			// Mover 2, pozycja odkładania		// przycisk monostabilny
	
//-------------------------------------------------------------------------------------------------------------------------------------------------------------------	
	//Sorter nasadek, CapPreScrewer	
	iCapSorterPreScrewerState							: INT;			// Stan
	sCapSorterPreScrewerState							: STRING;       // Stan
	lrCapSorterPreScrewerYAxisCVShow					: LREAL;		// Pozycja kartezjana oś Y
	lrCapSorterPreScrewerZAxisCVShow					: LREAL;		// Pozycja kartezjana oś Z
	lrCapSorterPreScrewerCAxisCVShow					: LREAL;		// Pozycja kartezjana oś C  
	bCapSorterPreScrewerHoming							: BOOL;			// Bazowanie					// Przycisk bistabilny 
	bCapSorterPreScrewerSetOffsetEncoderAxisZ			: BOOL;			// Ustaw offset encodera osi Z	//	Przycisk monostabilny
	bCapSorterPreScrewerPicker1Catch					: BOOL;			// Chwytak 1					// 	Przycisk bistabilny 
	bCapSorterPreScrewerPicker2Catch					: BOOL;			// Chwytak 2					// 	Przycisk bistabilny 
	bCapSorterPreScrewerPicker3Catch					: BOOL;			// Chwytak 3					// 	Przycisk bistabilny 
	bCapSorterPreScrewerPicker4Catch					: BOOL;			// Chwytak 4					// 	Przycisk bistabilny 
	bCapSorterPreScrewerPicker1Vacuum					: BOOL;			// Podsys 1						// 	Przycisk bistabilny 	
	bCapSorterPreScrewerPicker2Vacuum					: BOOL;			// Podsys 2						// 	Przycisk bistabilny 	
	bCapSorterPreScrewerPicker3Vacuum					: BOOL;			// Podsys 3						// 	Przycisk bistabilny 	
	bCapSorterPreScrewerPicker4Vacuum					: BOOL;			// Podsys 4						// 	Przycisk bistabilny 	
	bCapSorterPreScrewerPicker1Reject					: BOOL;			// Oddmuch 1					// 	Przycisk bistabilny	
	bCapSorterPreScrewerPicker2Reject					: BOOL;			// Oddmuch 2					// 	Przycisk bistabilny	
	bCapSorterPreScrewerPicker3Reject					: BOOL;			// Oddmuch 3					// 	Przycisk bistabilny	
	bCapSorterPreScrewerPicker4Reject					: BOOL;			// Oddmuch 4					// 	Przycisk bistabilny	
	
		//Kartezjan
	bCapSorterPreScrewerCartesianYForward				: BOOL;			// Y +							// Przycisk monostabilny
	bCapSorterPreScrewerCartesianYBackward				: BOOL;			// Y -							// Przycisk monostabilny
	bCapSorterPreScrewerCartesianZForward				: BOOL;			// Z +							// Przycisk monostabilny
	bCapSorterPreScrewerCartesianZBackward				: BOOL;			// Z -							// Przycisk monostabilny
	bCapSorterPreScrewerCartesianCForward				: BOOL;			// C +							// Przycisk monostabilny
	bCapSorterPreScrewerCartesianCBackward				: BOOL;			// C -							// Przycisk monostabilny
	                                                    	        	
		//Łapacz słomki    
 	lrCapSorterPreScrewerStrawCatcherCVShow				: LREAL;		// Pozycja łapacza słomek                           	
    bCapSorterPreScrewerStrawCatcherUp					: BOOL;			// Chwytaki do góry 			// Przycisk monostabilny
	bCapSorterPreScrewerStrawCatcherDown				: BOOL;			// Chwytaki do dołu 			// Przycisk monostabilny	
	bCapSorterPreScrewerStrawCatcherCatchOpen			: BOOL;			// Otwórz chwytaki słomek		// Przycisk bistabilny
	bCapSorterPreScrewerStrawCatcherCatchClose			: BOOL;			// Zamknij chwytaki słomek		// Przycisk bistabilny
	bCapSorterPreScrewerStrawCatcherActuatorIn			: BOOL;			//  Wsuń łapacz słomek			// Przycisk bistabilny
	bCapSorterPreScrewerStrawCatcherActuatorOut			: BOOL;			//  Wysuń łapacz słomek			// Przycisk bistabilny
                                                    	

                                                		
		//Podnośnik stacji wkladania nakrętek       		            	 
	bCapSorterPreScrewerCatcherStationUp					: BOOL;			// Stacja do góry 				// Przycisk monostabilny
	bCapSorterPreScrewerCatcherStationDown					: BOOL;			// Stacja do dołu 				// Przycisk monostabilny                 			
	bCapSorterPreScrewerBottleCatcherCatch					: BOOL;			// Chwytaki Butelek				// Przycisk bistabilny	
	lrCapSorterPreScrewerCatcherStationHeightCV				: LREAL;		// Aktualna wysokość chwytaka
	bCapSorterPreScrewerCatcherStationHeightSet				: BOOL;			// Ustaw pozycje				// Przycisk bistabilny
	bCapSorterPreScrewerBottleCatchOpenCalibration			: BOOL;			// Kalibruj otwarcie			// Przycisk bistabilny
	bCapSorterPreScrewerBottleCatchCloseCalibration			: BOOL;			// Kalibruj zamknięcie			// Przycisk bistabilny
	bCapSorterPreScrewerNextStep							: BOOL;			// Kolejny krok w serwice mode
                                                                        
	//Chwytak szyjki butelki pod wkladaczem nakrentek 1234                  
	bCapSorterPreScrewerCatchStationHoming	      			: BOOL;			// [H] Homing  					// Przycisk bistabilny	
	lrCapSorterPreScrewerCatchStationHeightSVShow			: LREAL;  		// Pozycja chwytaka
	bCapSorterPreScrewerManualBottleCatcherCatch			: BOOL;											// Przycisk bistabilny	        
 	
	
	bCapSorterManualVacuumPump								: BOOL; 
	// 1-Fliptop (prosta scieżka), 2-Pompka/Atomizer (Stawianie do pionu), 3-Fliptop z boku (stawianie do pionu + detekcja obróconej)
	AsCapSorterProductType									: ARRAY [1..10] OF STRING;
//	iCapSorterProductType									: INT;
	//
	AsCapSorterIndexShow									: ARRAY [1..30] OF STRING;	
//	uiCapSorterIndexShow									: UDINT;
	

	bCapSorterFeederAdvancedHoming							: BOOL;			// Bazowanie wózków "na zderzak"	
	bCapSorterPreScrewerAdvancedHoming						: BOOL;			// Bazowanie zaawansowane dotyczy osi Y
	
//-----------------------------------------------------------------------------------------------------------------------------------------------------

	bCapSorterCalculateParameters							: BOOL;			//	Oblicz paramaretry maszyny	//przycisk monostabilny
	bCapSorterSpare1										: BOOL;			//Rezerwa 1
	bCapSorterSpare2										: BOOL;			//Rezerwa 2
	bCapSorterSpare3										: BOOL;			//Rezerwa 3
	bCapSorterSpare4										: BOOL;			//Rezerwa 4
	bCapSorterSpare5										: BOOL;			//Rezerwa 5
	bCapSorterSpare6										: BOOL;			//Rezerwa 6
	bCapSorterSpare7										: BOOL;			//Rezerwa 7
	
	fbAlarms 											:FB_Events;	

	
END_VAR

// ---- POUs/MAIN.TcPOU
PROGRAM MAIN
VAR
END_VAR

gvl.iRunningMode;
gvl_checks.dCheckBounds;
gvl_communication.bChooseRecipe;
gvl_errorHandling.bError;
gvl_io.IbAirSupplyOK;
gvl_recipe.bCapSorterBrush1OnWheelEnableShow;
gvl_standaloneunit.bChooseRecipe;
gvl_vis.AsCapSorterIndexShow;

END_PROGRAM

// ---- POUs/FB_DigitalInput.TcPOU
//==================================================================================================
//							Beckhoff Automation Poland
//									14.03.2023
//
// Code owner: TG
//
// Function block for processing digital inputs. 
// Includes filters, simulating and edges detection.
//
// Used libraries: 
//	Tc2_standard						|| 3.3.3.0
//
// Used FBs:
//
// Used DUTs:
//
//  v1.0	|| TC v 3.1.4024.40		|| First edition
//==================================================================================================
FUNCTION_BLOCK FB_DigitalInput

VAR_INPUT
	In 						AT %I* 				: BOOL;
END_VAR

VAR
	
	bManual										: BOOL;	 // HMI
	bManualIn									: BOOL;	 // HMI
	{attribute 'hide'}
	_bCheckFS									: BOOL;
	{attribute 'hide'}
	_bIn	 									: BOOL;
	{attribute 'hide'}
	_bInRE										: BOOL;
	{attribute 'hide'}
	_bInFE										: BOOL;
	{attribute 'hide'}
	_tTimeOn									: TIME;
	{attribute 'hide'}
	_tTimeOff									: TIME;	
	{attribute 'hide'}
	_tTimeFS									: TIME;
	{attribute 'hide'}
	TimeFS										: TOF;	
	{attribute 'hide'}
	rtTrigger									: R_TRIG;
	{attribute 'hide'}
	ftTrigger									: F_TRIG;
END_VAR

{attribute 'monitoring' := 'variable'}
PROPERTY bCheckFS								: BOOL
GET
bCheckFS										:= _bCheckFS;
END_GET
SET
_bCheckFS										:= bCheckFS;
END_SET
END_PROPERTY

{attribute 'monitoring' := 'variable'}
PROPERTY bErrFS 								: BOOL							//Fail-safe error
GET
bErrFS											:= NOT TimeFS.Q AND bCheckFS;
END_GET
END_PROPERTY

{attribute 'monitoring' := 'variable'}
PROPERTY bIn 									: BOOL							//Processed input variable
GET
bIn												:= _bIn;
END_GET
SET
_bIn											:= bIn;
END_SET
END_PROPERTY

{attribute 'monitoring' := 'variable'}
PROPERTY bInFE 									: BOOL							//Falling edge detected
GET
bInFE											:= ftTrigger.Q;
END_GET
END_PROPERTY

{attribute 'monitoring' := 'variable'}
PROPERTY bInRE 									: BOOL							//Rising edge detected
GET
bInRE											:= rtTrigger.Q;
END_GET
END_PROPERTY

METHOD Filter 									: BOOL							//Activation and disable filter
VAR_INST
	{attribute 'hide'}
	TimeON										: TON;
	{attribute 'hide'}
	TimeOFF										: TOF;	
END_VAR
TimeON(IN := In, PT := tTimeON);
TimeOFF(IN := TimeON.Q, PT := tTimeOff);

bIn												:= TimeOFF.Q;
END_METHOD

METHOD FilterTrig 								: BOOL						//Activation and disable filter with edges detection
Filter();		
RTrig();
FTrig();
END_METHOD

METHOD FS 										: BOOL								// Fail-safe detection timer
VAR_INST
	{attribute 'hide'}
	bLastIn										: BOOL;	
END_VAR
TimeFS(IN := bLastIn <> In, PT := tTimeFS);	

bLastIn											:= In;
END_METHOD

METHOD PRIVATE FTrig 							: BOOL							// Falling edge detection
ftTrigger(CLK := bIn);
END_METHOD

METHOD Manual 									: BOOL							//Manually controlled input
IF bManual THEN
	ManualEx(bIn := bManualIn);
END_IF
END_METHOD

METHOD ManualEx 									: BOOL							//Manually controlled input
VAR_INPUT
	bIn												: BOOL;
END_VAR
bCheckFS										:= FALSE;
bIn												:= bIn;
END_METHOD

METHOD ManualExTrig 								: BOOL						//Manually controlled input with edges detection
VAR_INPUT
	bManual											: BOOL;
	bIn												: BOOL;
END_VAR
ManualEx(bIn := bManualIn);		
RTrig();
FTrig();
END_METHOD

METHOD ManualTrig 								: BOOL						//Manually controlled input with edges detection
Manual();		
RTrig();
FTrig();
END_METHOD

METHOD Raw 										: BOOL							// Raw value
bIn												:= In;
END_METHOD

METHOD PRIVATE RTrig 							: BOOL							//Rising edge detection
rtTrigger(CLK := bIn);
END_METHOD

{attribute 'monitoring' := 'variable'}
PROPERTY tTimeFS 								: TIME							//fail-safe control time [ms]
GET
tTimeFS											:= _tTimeFS;
END_GET
SET
_tTimeFS										:= tTimeFS;
END_SET
END_PROPERTY

{attribute 'monitoring' := 'variable'}
PROPERTY tTimeOff 								: TIME						//disabling filter time [ms]
GET
tTimeOff										:= _tTimeOff;
END_GET
SET
_tTimeOff										:= tTimeOff;
END_SET
END_PROPERTY

{attribute 'monitoring' := 'variable'}
PROPERTY tTimeOn 								: TIME							//activation delay time [ms]
GET
tTimeOn											:= _tTimeOn;
END_GET
SET
_tTimeOn									:= tTimeOn;
END_SET
END_PROPERTY

END_FUNCTION_BLOCK

// ---- POUs/FB_DigitalOutput.TcPOU
//==================================================================================================
//							Beckhoff Automation Poland
//									14.03.2023
//
// Code owner: TG
//
// Function block for processing digital outputs. 
// Includes filters, simulating, various operational modes selection and edges detection.
//
// Used libraries: 
//	Tc2_standard						|| 3.3.3.0
//
// Used FBs:
//
// Used DUTs:
//
//  v1.0	|| TC v 3.1.4024.40		|| First edition
//==================================================================================================
FUNCTION_BLOCK FB_DigitalOutput
VAR
	Out 					AT %Q* 				: BOOL;
	bManualIn									: BOOL;		// HMI
	
	{attribute 'hide'}
	bManualMode_Internal						: BOOL;		// Internal flag - active when manual mode selected
	_bIn										: BOOL;
	{attribute 'hide'}
	_bOut										: BOOL; 
	{attribute 'hide'}
	_tTimeDelay									: TIME;
	{attribute 'hide'}
	_tTimeOn									: TIME;
	{attribute 'hide'}
	_tTimeOff									: TIME;
	{attribute 'hide'}
	_nMode										: DINT;															
END_VAR

CASE nMode OF							//case regarding mode selection 

	0:	// false
		Off();
	
	1:	// true
		On();

	2:	// auto normal
		Auto();
		
	9:	// manual
		Manual();
	
	10:	// clock
		Clock();

	11: // min OFF, min ON	
		MinOnOff();	
	
	20: // single TP
		SingleTP();
	
	21: // single TON
		SingleTON();	
							
	30: // mutli TP
		MultiTP();

	31:	// mutli TON
		MultiTON();
		
ELSE		
	Off();
	
		
END_CASE;

METHOD Auto 									: BOOL							//output actual value 
VAR_INPUT
END_VAR
bOut											:= bIn;

bManualMode_Internal							:= FALSE;
END_METHOD

PROPERTY bIn 									: BOOL								//value before processing
GET
bIn												:=_bIn;
END_GET
SET
_bIn											:= bIn;
END_SET
END_PROPERTY

PROPERTY bOut 									: BOOL							//processed output value
GET
bOut											:= _bOut;
END_GET
SET
_bOut											:= bOut;
Out												:= bOut;
END_SET
END_PROPERTY

METHOD Clock 									: BOOL							//use output for specifed time with pause between
VAR_INST
	{attribute 'hide'}
	tonTimer									: TON;
END_VAR
tonTimer(IN := NOT tonTimer.Q,
		PT										:= tTimeOn + tTimeOff);
bOut											:= tonTimer.ET <  tTimeOn;
		
bManualMode_Internal							:= FALSE;
END_METHOD

METHOD Manual 									: BOOL							//Control output value manually
IF bManualMode_Internal THEN
	bOut										:= bManualIn;
ELSE
	bManualIn									:= bOut;
END_IF

bManualMode_Internal							:= TRUE;
END_METHOD

METHOD ManualEx 								: BOOL							//Control output value manually
VAR_INPUT
	bIn											: BOOL;
END_VAR
bOut											:= bIn;

bManualMode_Internal							:= FALSE;
END_METHOD

METHOD MinOnOff 								: BOOL						//output with specific active and disabled time
VAR_INST
	TimeMinOn									: TON;
	TimeMinOff									: TON;	
END_VAR
TimeMinOff(IN := NOT bOut, PT := tTimeOff);			
                        						
TimeMinOn(IN := bOut, PT := tTimeOn);	
		
IF TimeMinOn.Q THEN
	bOut										:= bIn;
END_IF;			
		
IF TimeMinOff.Q THEN
	bOut										:= bIn;
END_IF;

bManualMode_Internal							:= FALSE;
END_METHOD

METHOD MultiTON 								: BOOL						//activation delay dependent from value
VAR_INST
	Timer										: TON;
END_VAR
Timer(IN := bIn, PT := tTimeDelay);

bOut											:= Timer.Q;

bManualMode_Internal							:= FALSE;
END_METHOD

METHOD MultiTP 									: BOOL							//pulse dependent from value
VAR_INST
	Timer										: TP;
END_VAR
Timer(IN := bIn, PT := tTimeOn);
		
bOut											:= Timer.Q;

bManualMode_Internal							:= FALSE;
END_METHOD

PROPERTY nMode 									: DINT							//mode selection value: 0- false 1-true 2 - auto_normal, 10- clock, 20 - single tp, 21 - single ton, 9 - manual, 30 - multi tp, 31 - multi ton, 11 - min ON, min OFF
GET
nMode											:= _nMode;
END_GET
SET
_nMode											:= nMode;
END_SET
END_PROPERTY

METHOD Off 										: BOOL								//set value FALSE
bOut											:= FALSE;

bManualMode_Internal							:= FALSE;
END_METHOD

METHOD On 										: BOOL								//set value TRUE
bOut											:= TRUE;

bManualMode_Internal							:= FALSE;
END_METHOD

METHOD SingleTON 								: BOOL						//activation delay 
VAR_INST
	Timer										: TON;
END_VAR
Timer(IN := TRUE, PT := tTimeDelay);

bOut											:= Timer.Q;

bManualMode_Internal							:= FALSE;
END_METHOD

METHOD SingleTP 								: BOOL						//single pulse
VAR_INST
	Timer										: TP;
END_VAR
Timer(IN := TRUE, PT := tTimeOn);

bOut											:= Timer.Q;

bManualMode_Internal							:= FALSE;
END_METHOD

PROPERTY tTimeDelay  								: TIME						//delay time in [ms], for Single/MultiTON mode
GET
tTimeDelay										:= _tTimeDelay;
END_GET
SET
_tTimeDelay										:= tTimeDelay;
END_SET
END_PROPERTY

PROPERTY tTimeOff 								: TIME						//minimum output on time [ms], for minOnOff mode
GET
tTimeOff										:= _tTimeOff;
END_GET
SET
_tTimeOff										:= tTimeOff;
END_SET
END_PROPERTY

PROPERTY tTimeOn 								: TIME						//minimum output off time [ms], for minOnOff mode
GET
tTimeOn											:=_tTimeOn;
END_GET
SET
_tTimeOn										:= tTimeOn;
END_SET
END_PROPERTY

END_FUNCTION_BLOCK
